# EPICS substitutions: db/Beckhoff_2XXX/ecmcEL2612.substitutions
file "ecmc_binaryOutput-chX.template"
{
  pattern {CH_ID}
          {01   }
          {02   }
}
